FUNCTION_BLOCK FB_SSI_Encoder
VAR_INPUT
	
	ValueIn		: UDINT;				(* Analog input value *)
	MinIn		: UDINT;				(* Minimum value for input signal *)
	MaxIn		: UDINT;				(* Maximum value for input signal *)
	MinOut		: REAL;					(* Minimum value for output signal *)
	MaxOut		: REAL;					(* Maximum value for output signal *)
	
END_VAR
VAR_OUTPUT
	Out			: SSI_Encoder ;
END_VAR
VAR
	RangeIn: REAL;
	RangeOut: REAL;
END_VAR

(* Rescale input *)

	RangeIn 			:= UDINT_TO_REAL( MaxIn ) - UDINT_TO_REAL( MinIn );

	RangeOut 			:= MaxOut - MinOut;

	IF RangeIn <> 0
	(*  AND ValueIn >= MinIn
	  AND ValueIn <= MaxIn *) THEN
		Out.rScaled 	:= ( ( ( UDINT_TO_REAL( ValueIn  -  MinIn ) ) / RangeIn ) * RangeOut ) + MinOut;
	ELSE
		Out.rScaled		:= 0;
	END_IF

	Out.uCounterValue			:= ValueIn;

END_FUNCTION_BLOCK

(* stored: Version 1.1.0.1, ProductVersion 3.1.4024.12
   POU FB_SSI_Encoder: Id {c3d21860-8721-40ff-8390-26b599d8444b}, SpecialFunc None *)
